Staubli VAL3: decTrajPt.pgx

public program decTrajPt(bool& x_bFlag)
  local num l_nIndex
  local num l_nRetVal
begin
  // Copyright (c) 2016, Ocado Technology - Robotics Research Team
  //
  // Licensed under the Apache License, Version 2.0 (the "License");
  // you may not use this file except in compliance with the License.
  // You may obtain a copy of the License at
  //
  //     http://www.apache.org/licenses/LICENSE-2.0
  //
  // Unless required by applicable law or agreed to in writing, software
  // distributed under the License is distributed on an "AS IS" BASIS,
  // WITHOUT WARRANTIES OR CONDITIONS OF ANY KIND, either express or implied.
  // See the License for the specific language governing permissions and
  // limitations under the License.



  // decode message ID 11 body (data)

  // assume failure to decode
  rosTrajPtAck.header.nReplyCode=2

  // sequence
  l_nRetVal=fromBinary(rosTrajPtMsg.body.nData,4,"-4l",rosTrajPtMsg.jointTrajPt.nSeq)
  if (l_nRetVal!=1)
    x_bFlag=false
    return
  endIf

  // joints[10]
  for l_nIndex=0 to 9 step 1
    l_nRetVal=fromBinary(rosTrajPtMsg.body.nData[(l_nIndex*4)+4],4,"4.0l",rosTrajPtMsg.jointTrajPt.nJoints[l_nIndex])
    if (l_nRetVal!=1)
      x_bFlag=false
      return
    endIf
  endFor

  // velocity
  l_nRetVal=fromBinary(rosTrajPtMsg.body.nData[44],4,"4.0l",rosTrajPtMsg.jointTrajPt.nVelocity)
  if (l_nRetVal!=1)
    x_bFlag=false
    return
  endIf

  // duration
  l_nRetVal=fromBinary(rosTrajPtMsg.body.nData[48],4,"4.0l",rosTrajPtMsg.jointTrajPt.nDuration)
  if(l_nRetVal!=1)
    x_bFlag=false
    return
  endIf

  // decoding successful
  rosTrajPtAck.header.nReplyCode=1
  rosTrajPtAck.jointTrajPt.nSeq=rosTrajPtMsg.jointTrajPt.nSeq
  nTotalTrajPoint = nTotalTrajPoint + rosTrajPtMsg.jointTrajPt.nSeq+1
  x_bFlag=true
end
